(* Schneider Machine Expert - Basic project Timer 2, file version 1.7.0.0 *)
(* ProjectInformations: Name=New project *)

HARDWARE
  Cpu 0: TM221M16R/G
  EthernetConfiguration: NetworkName=M221, IpAllocationMode=FixedAddress, IpAddress=0.0.0.0, SubnetMask=0.0.0.0
  SerialLineConfiguration: Baud=Baud19200, Parity=ParityEven, DataBits=DataBits8, StopBits=StopBits1, PhysicalMedium=PhysicalMediumRs485, TransmissionMode=TransmissionModeModbusRtu, SlaveId=1, Addressing=SlaveAddressing
  MastTask: UsePeriodScanMode=false, PeriodScan=100
  FastTask: Period=255
  CpuBehavior: StartingMode=StartAsPreviousState, AutoSaveRamOnEeprom=true, WatchdogPeriod=250

SYMBOLS  (address, symbol, comment, settings)
  %TM0        "T1 3""  [Preset=3, Base=OneSecond]
  %TM1        "T2 3""  [Preset=3, Base=OneSecond]
  %I0.0       "Auto"
  %I0.1       "Manual"
  %I0.2       "S1"
  %I0.3       "S2"
  %Q0.0       "P1"
  %Q0.1       "P2"

POU New POU
  (* SectionNumber=1 *)

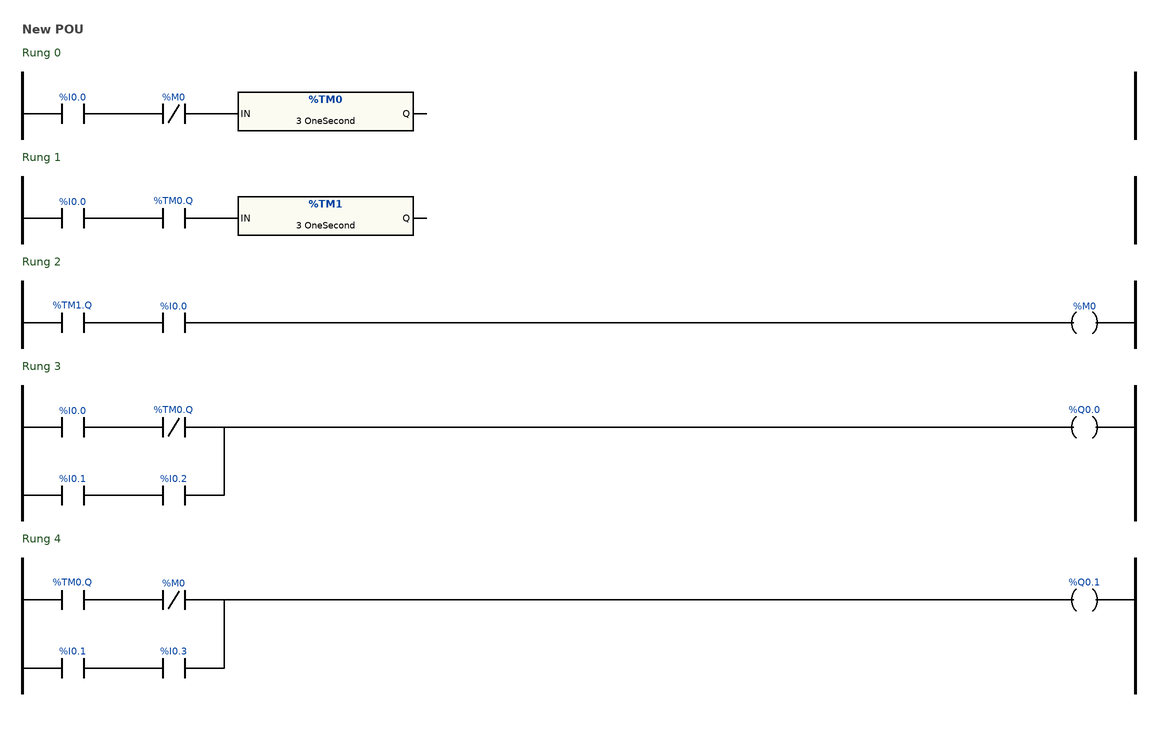

// Rung 0
  BLK %TM0
  LD %I0.0
  ANDN %M0
  IN
  END_BLK
  // as ST:
  //   %TM0(IN := %I0.0 AND NOT %M0);

// Rung 1
  BLK %TM1
  LD %I0.0
  AND %TM0.Q
  IN
  END_BLK
  // as ST:
  //   %TM1(IN := %I0.0 AND %TM0.Q);

// Rung 2
  LD %TM1.Q
  AND %I0.0
  ST %M0
  // as ST:
  //   %M0 := %TM1.Q AND %I0.0;

// Rung 3
  LD %I0.0
  ANDN %TM0.Q
  OR( %I0.1
  AND %I0.2
  )
  ST %Q0.0
  // as ST:
  //   %Q0.0 := %I0.0 AND NOT %TM0.Q OR %I0.1 AND %I0.2;

// Rung 4
  LD %TM0.Q
  ANDN %M0
  OR( %I0.1
  AND %I0.3
  )
  ST %Q0.1
  // as ST:
  //   %Q0.1 := %TM0.Q AND NOT %M0 OR %I0.1 AND %I0.3;
